{attribute 'linkalways'} 
{attribute 'no_explicit_call' := 'This FB is a CLASS and must be accessed using methods or properties'}
{attribute 'enable_dynamic_creation'}
FUNCTION_BLOCK FINAL ABS_SINT EXTENDS Node
VAR
	in : _SINT(0);
	out : _SINT(0);
END_VAR

METHOD PUBLIC Clone : I_Node
VAR
	pNode : POINTER TO ABS_SINT;
END_VAR
pNode := __NEW(ABS_SINT);
Clone := pNode^;
END_METHOD

METHOD FB_init : BOOL
VAR_INPUT
	bInitRetains : BOOL; // if TRUE, the retain variables are initialized (warm start / cold start)
	bInCopyCode : BOOL;  // if TRUE, the instance afterwards gets moved into the copy code (online change)
END_VAR
AddInput('in',THIS^.in);
AddOutput('out', THIS^.out);
END_METHOD

METHOD PROTECTED OnExecute
VAR
END_VAR
out.Value := ABS(in.Value);
END_METHOD

END_FUNCTION_BLOCK

(* stored: Version 1.1.0.1, ProductVersion 3.1.4024.15
   POU ABS_SINT: Id {ef10e9ac-0cac-4f3c-9bce-0a3194610773}, SpecialFunc None
   Folder Constructor: Id {2e49a862-3915-48db-b962-0f0148f8f0a2}
   Method Clone: Id {6f0839fc-cada-421f-9a99-f9d61bbd5154}
   Method FB_init: Id {0778e262-9e69-414c-a8ca-5a315fa88b7c}
   Method OnExecute: Id {70e9c3c6-3502-405b-b3a7-8eb4909e1ee3} *)
